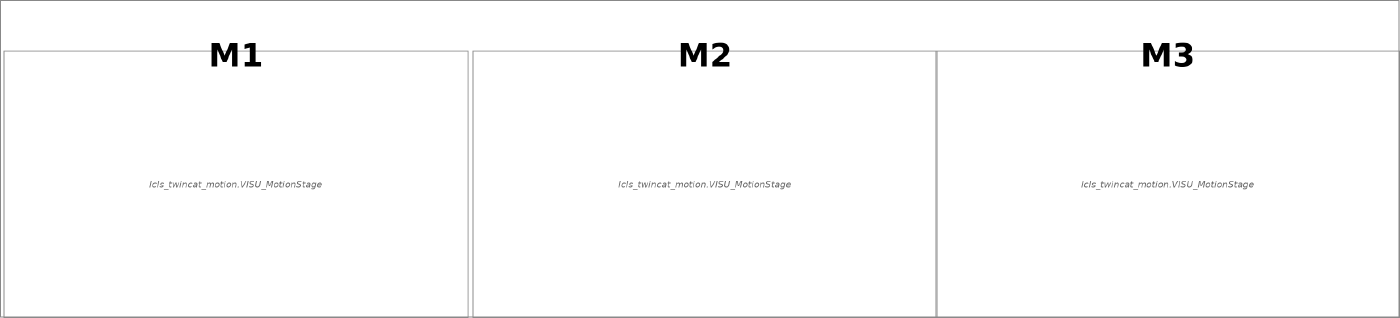
VISUALIZATION Visualization  // 1567x357
    Frame (4,57 520x300)
        shows lcls_twincat_motion.VISU_MotionStage(VisuMotionStage := Main.M1, Extras := Main.stM1Extra)
    Label (189,47 150x30), "M1"
    Frame (529,57 520x300)
        shows lcls_twincat_motion.VISU_MotionStage(VisuMotionStage := Main.M2, Extras := Main.stM2Extra)
    Label (714,47 150x30), "M2"
    Frame (1047,57 520x300)
        shows lcls_twincat_motion.VISU_MotionStage(VisuMotionStage := Main.M3, Extras := Main.stM3Extra)
    Label (1232,47 150x30), "M3"
END_VISUALIZATION

(* stored: Version 1.1.0.1, ProductVersion 3.1.4024.4
   Visu Visualization: Id {46038cbc-714f-4f35-b697-7f366f8e7109} *)
